FUNCTION "Ventilstatus" : Void
{ S7_Optimized_Access := 'TRUE' }
VERSION : 0.1
   VAR_INPUT 
      SRM_auf : Bool;
      SRM_zu : Bool;
      A_Ventil : Bool;
      Zeit : Time;
   END_VAR

   VAR_OUTPUT 
      "Farbe HMI" : USInt;   // 0: geschlossen (grau) 1: geöffnet (grün) 2: Störung (rot)
      Mld_TO_oeffnen : Bool;
      Mld_TO_schliessen : Bool;
   END_VAR

   VAR_IN_OUT 
      TO_oeffnen {InstructionName := 'TON_TIME'; LibVersion := '1.0'} : TON_TIME;
      TO_schliessen {InstructionName := 'TON_TIME'; LibVersion := '1.0'} : TON_TIME;
      Mld_Sensorfehler : Bool;
   END_VAR

   VAR CONSTANT 
      grau : USInt;
      grün : USInt := 1;
      rot : USInt := 2;
   END_VAR


BEGIN
	// Beide an
	IF #SRM_auf AND #SRM_zu THEN
	    #Mld_Sensorfehler := TRUE;
	ELSIF "DB_ANLAGE".IN.Quitt_Err THEN
	    #Mld_Sensorfehler := FALSE;
	END_IF;
	
	// Zeitüberschreitung öffnen
	#TO_oeffnen(IN := #A_Ventil AND NOT #SRM_auf,
	            PT:= #Zeit,
	            Q=> #Mld_TO_oeffnen);
	
	// Zeitüberschreitung schließen
	#TO_schliessen(IN := NOT #A_Ventil AND NOT #SRM_zu,
	            PT := #Zeit,
	            Q => #Mld_TO_schliessen);
	
	//--> Visu
	IF #Mld_TO_oeffnen OR #Mld_TO_schliessen OR #Mld_Sensorfehler THEN
	    #"Farbe HMI" := #rot;
	ELSIF #A_Ventil THEN
	    #"Farbe HMI" := #grün;
	ELSE
	    #"Farbe HMI" := #grau;
	END_IF;
END_FUNCTION

FUNCTION "Ventilstatus_einfach" : Void
{ S7_Optimized_Access := 'TRUE' }
VERSION : 0.1
   VAR_INPUT 
      A_Ventil : Bool;
   END_VAR

   VAR_OUTPUT 
      "Farbe HMI" : USInt;   // 0: geschlossen (grau) 1: geöffnet (grün) 2: Störung (rot)
   END_VAR

   VAR CONSTANT 
      grau : USInt;
      grün : USInt := 1;
      rot : USInt := 2;
   END_VAR


BEGIN
	//--> Visu
	IF #A_Ventil THEN
	    #"Farbe HMI" := #grün;
	ELSE
	    #"Farbe HMI" := #grau;
	END_IF;
END_FUNCTION

DATA_BLOCK "Deckel_CM01"   // DB1190
// stored: AutoNumber false, InstanceOfName Deckel, InstanceOfType FB
"Deckel"
BEGIN
END_DATA_BLOCK

DATA_BLOCK "Deckel_CM02"   // DB1191
// stored: AutoNumber false, InstanceOfName Deckel, InstanceOfType FB
"Deckel"
BEGIN
END_DATA_BLOCK

DATA_BLOCK "Uhrzeit"   // DB8
// stored: AutoNumber false, InstanceOfName Uhrzeit_WSU, InstanceOfType FB
"Uhrzeit_WSU"
BEGIN
END_DATA_BLOCK

DATA_BLOCK "DI_FU_Fahrt"   // DB181
// stored: AutoNumber false, InstanceOfName FB_FU_OUT_TW, InstanceOfType FB
"FB_FU_OUT_TW"
BEGIN
END_DATA_BLOCK

DATA_BLOCK "DI_FU_Hub_links"   // DB182
// stored: AutoNumber false, InstanceOfName FB_FU_OUT_TW, InstanceOfType FB
"FB_FU_OUT_TW"
BEGIN
END_DATA_BLOCK

DATA_BLOCK "DI_FU_Hub_rechts"   // DB183
// stored: AutoNumber false, InstanceOfName FB_FU_OUT_TW, InstanceOfType FB
"FB_FU_OUT_TW"
BEGIN
END_DATA_BLOCK

DATA_BLOCK "DI_FU_WR02"   // DB184
// stored: AutoNumber false, InstanceOfName FB_FU_OUT_TW, InstanceOfType FB
"FB_FU_OUT_TW"
BEGIN
END_DATA_BLOCK

DATA_BLOCK "DI_FU_WR03"   // DB185
// stored: AutoNumber false, InstanceOfName FB_FU_OUT_TW, InstanceOfType FB
"FB_FU_OUT_TW"
BEGIN
END_DATA_BLOCK

DATA_BLOCK "DI_FW_1"   // DB11
AUTHOR : MS
VERSION : 0.0
// stored: AutoNumber false, InstanceOfName FB_FW_x, InstanceOfType FB
"FB_FW_x"
BEGIN
   Micro.Adr_UP[1] := 16#0066;
   Micro.Adr_UP[2] := 16#006A;
   Micro.Adr_UP[3] := 16#006E;
   Micro.Adr_UP[4] := 16#0077;
   Micro.Adr_UP[5] := 16#007D;
   Micro.Adr_UP[6..13] := 16#0086;
   Micro.Adr_UP[14] := 16#0082;
   Micro.Adr_UP[15] := 16#0084;
   Micro.Liste[0] := 16#02;
   Micro.Liste[1] := 16#14;
   Micro.Liste[2] := 16#05;
   Micro.Liste[3] := 16#00;
   Micro.Liste[4] := 16#03;
   Micro.Liste[5] := 16#14;
   Micro.Liste[6] := 16#05;
   Micro.Liste[7] := 16#00;
   Micro.Liste[8] := 16#01;
   Micro.Liste[9] := 16#15;
   Micro.Liste[10] := 16#04;
   Micro.Liste[11] := 16#0E;
   Micro.Liste[12] := 16#18;
   Micro.Liste[13] := 16#16;
   Micro.Liste[14] := 16#0B;
   Micro.Liste[15] := 16#19;
   Micro.Liste[16] := 16#00;
   Micro.Liste[17] := 16#09;
   Micro.Liste[18] := 16#10;
   Micro.Liste[19] := 16#03;
   Micro.Liste[20] := 16#07;
   Micro.Liste[21] := 16#0C;
   Micro.Liste[22] := 16#00;
   Micro.Liste[23] := 16#14;
   Micro.Liste[24] := 16#09;
   Micro.Liste[25] := 16#11;
   Micro.Liste[26] := 16#12;
   Micro.Liste[27] := 16#00;
   Micro.Liste[28] := 16#0A;
   Micro.Liste[29] := 16#00;
   Micro.Liste[30] := 16#06;
   Micro.Liste[31..79] := 16#00;
END_DATA_BLOCK

DATA_BLOCK "DI_FW_Auftrag_DB"   // DB9
// stored: AutoNumber false, InstanceOfName FB_FW_Auftrag, InstanceOfType FB
"FB_FW_Auftrag"
BEGIN
END_DATA_BLOCK

DATA_BLOCK "DI_FW_HUB_links"   // DB22
AUTHOR : MS
// stored: AutoNumber false, InstanceOfName FB_HUB_FW_li, InstanceOfType FB
"FB_HUB_FW_li"
BEGIN
END_DATA_BLOCK

DATA_BLOCK "DI_FW_HUB_rechts"   // DB23
AUTHOR : MS
// stored: AutoNumber false, InstanceOfName FB_HUB_FW_re, InstanceOfType FB
"FB_HUB_FW_re"
BEGIN
END_DATA_BLOCK

DATA_BLOCK "DI_FW_MANAGER"   // DB10
AUTHOR : MS
// stored: AutoNumber false, InstanceOfName FB_FW_MANAGER, InstanceOfType FB
"FB_FW_MANAGER"
BEGIN
   Kettenpos[1..4] := 16#00;
   FW_DAT[1..20].WT_NR_LANG := 0;
   FW_DAT[1].IST_POS := 16#02;
   FW_DAT[2].IST_POS := 16#0B;
   FW_DAT[3].IST_POS := 16#2C;
   FW_DAT[4].IST_POS := 16#4A;
   FW_DAT[5].IST_POS := 16#02;
   FW_DAT[6].IST_POS := 16#2F;
   FW_DAT[7..20].IST_POS := 16#00;
   FW_DAT[1..20].ZIEL_POS := 16#00;
   FW_DAT[1..20].Fahrt_Vor := FALSE;
   FW_DAT[1..20].Fahrt_Rck := FALSE;
   FW_DAT[1..20].Heben := FALSE;
   FW_DAT[1..20].Senken := FALSE;
   FW_DAT[1..6].Bereit := TRUE;
   FW_DAT[7..20].Bereit := FALSE;
   FW_DAT[1..20].Fehler := FALSE;
   FW_DAT[1..20].Dummy := FALSE;
   FW_DAT[1..20].res := FALSE;
   FW_DAT[1..20].Tipp := FALSE;
   FW_DAT[1..6].Hand := TRUE;
   FW_DAT[7..20].Hand := FALSE;
   FW_DAT[1..20].Auto_Stop := FALSE;
   FW_DAT[1..20].Auto := FALSE;
   FW_DAT[1..20].Halt := FALSE;
   FW_DAT[1..6].K_Auto := TRUE;
   FW_DAT[7..20].K_Auto := FALSE;
   FW_DAT[1..4].Kette_wait_Start := TRUE;
   FW_DAT[5..20].Kette_wait_Start := FALSE;
   FW_DAT[1..4].Kette_wait_Ende := TRUE;
   FW_DAT[5..20].Kette_wait_Ende := FALSE;
   FW_DAT[1..4].Unten := TRUE;
   FW_DAT[5..20].Unten := FALSE;
   FW_DAT[1..20].Z_Sensor := FALSE;
   FW_DAT[1..20].Oben := FALSE;
   FW_DAT[1..6].mittig := TRUE;
   FW_DAT[7..20].mittig := FALSE;
   FW_DAT[1..20].HWmittig := FALSE;
   FW_DAT[1..20].res_7 := FALSE;
   FW_DAT[1..20].res_8 := FALSE;
   FW_DAT[1..20].res_9 := FALSE;
   FW_DAT[1..20].WT_DB_Nr := 16#00;
   FW_DAT[1].IstInc := 1998;
   FW_DAT[2].IstInc := 10998;
   FW_DAT[3].IstInc := 43999;
   FW_DAT[4].IstInc := 49759;
   FW_DAT[5..20].IstInc := 0;
   FW_DAT[1..20].Stangen_Nr := 16#00;
   FW_DAT[1..20].WT_Typ := 16#00;
   FW_DAT[1..20].priorisirt := FALSE;
   FW_DAT[1..20].in_Anlage := FALSE;
   FW_DAT[1..20].in_Entmetall := FALSE;
   FW_DAT[1..20].aus_Anlage := FALSE;
   FW_DAT[1..20].aus_Entmetall := FALSE;
   FW_DAT[1..20].Speicherprog := FALSE;
   FW_DAT[1..20].Trommel := FALSE;
   FW_DAT[1..20].Leer_WT := FALSE;
   FW_DAT[1..20].BefX := 16#00;
END_DATA_BLOCK

DATA_BLOCK "DI_FW_POS_1"   // DB21
// stored: AutoNumber false, InstanceOfName FB_POS_FW_INC, InstanceOfType FB
"FB_POS_FW_INC"
BEGIN
END_DATA_BLOCK

DATA_BLOCK "DI_QF_WR02_03"   // DB31
// stored: AutoNumber false, InstanceOfName FB_QF, InstanceOfType FB
"FB_QF"
BEGIN
END_DATA_BLOCK

DATA_BLOCK "Tor"   // DB1092
// stored: AutoNumber false, InstanceOfName RT, InstanceOfType FB
"RT"
BEGIN
END_DATA_BLOCK

DATA_BLOCK "TCON_DI"   // DB365
// stored: AutoNumber false, InstanceOfName TCON, OfSystemLibElement TCON, OfSystemLibVersion 4.0
"TCON"
   // VAR_INPUT
   //    REQ : Bool := TRUE;
   //    ID : CONN_OUC := 16#0002;
   // END_VAR
   // VAR_OUTPUT
   //    DONE : Bool := TRUE;
   //    BUSY : Bool := FALSE;
   //    ERROR : Bool := FALSE;
   //    STATUS : Word := 16#0000;
   // END_VAR
   // VAR_IN_OUT
   //    CONNECT : Variant;
   // END_VAR
BEGIN
END_DATA_BLOCK

DATA_BLOCK "TDISCON_DI"   // DB368
// stored: AutoNumber false, InstanceOfName T_DISCON, OfSystemLibElement TDISCON, OfSystemLibVersion 2.1
"T_DISCON"
   // VAR_INPUT
   //    REQ : Bool := FALSE;
   //    ID : CONN_OUC := 16#0000;
   // END_VAR
   // VAR_OUTPUT
   //    DONE : Bool := FALSE;
   //    BUSY : Bool := FALSE;
   //    ERROR : Bool := FALSE;
   //    STATUS : Word := 16#7000;
   // END_VAR
BEGIN
END_DATA_BLOCK

DATA_BLOCK "TRCV_DI"   // DB367
// stored: AutoNumber false, InstanceOfName TRCV, OfSystemLibElement TRCV, OfSystemLibVersion 4.0
"TRCV"
   // VAR_INPUT
   //    EN_R : Bool := TRUE;
   //    ID : CONN_OUC := 16#0002;
   //    LEN : UDInt := 30;
   //    ADHOC : Bool := FALSE;
   // END_VAR
   // VAR_OUTPUT
   //    NDR : Bool := TRUE;
   //    BUSY : Bool := FALSE;
   //    ERROR : Bool := FALSE;
   //    STATUS : Word := 16#0000;
   //    RCVD_LEN : UDInt := 30;
   // END_VAR
   // VAR_IN_OUT
   //    DATA : Variant;
   //    ADDR : Variant;
   // END_VAR
BEGIN
END_DATA_BLOCK

DATA_BLOCK "TSEND_DI"   // DB366
// stored: AutoNumber false, InstanceOfName TSEND, OfSystemLibElement TSEND, OfSystemLibVersion 4.0
"TSEND"
   // VAR_INPUT
   //    REQ : Bool := TRUE;
   //    ID : CONN_OUC := 16#0002;
   //    LEN : UDInt := 30;
   // END_VAR
   // VAR_OUTPUT
   //    DONE : Bool := TRUE;
   //    BUSY : Bool := FALSE;
   //    ERROR : Bool := FALSE;
   //    STATUS : Word := 16#0000;
   // END_VAR
   // VAR_IN_OUT
   //    DATA : Variant;
   //    ADDR : Variant;
   // END_VAR
BEGIN
END_DATA_BLOCK

DATA_BLOCK "FP_CM01.GP01"   // DB1001
// stored: AutoNumber false, InstanceOfName FP_Saeure.GP0x, InstanceOfType FB
"FP_Saeure.GP0x"
BEGIN
END_DATA_BLOCK

DATA_BLOCK "FP_CM02.GP04"   // DB1004
// stored: AutoNumber false, InstanceOfName FP_Saeure.GP0x, InstanceOfType FB
"FP_Saeure.GP0x"
BEGIN
END_DATA_BLOCK

DATA_BLOCK "Pu_CL01.GP08"   // DB1008
// stored: AutoNumber false, InstanceOfName Pu_Entl.GP0x, InstanceOfType FB
"Pu_Entl.GP0x"
BEGIN
END_DATA_BLOCK

DATA_BLOCK "Pu_CL02.GP09"   // DB1009
// stored: AutoNumber false, InstanceOfName Pu_Entl.GP0x, InstanceOfType FB
"Pu_Entl.GP0x"
BEGIN
END_DATA_BLOCK

DATA_BLOCK "Pu_CM05.GP11_DB"   // DB1011
// stored: AutoNumber false, InstanceOfName Pu_CM05.GP11, InstanceOfType FB
"Pu_CM05.GP11"
BEGIN
END_DATA_BLOCK

DATA_BLOCK "Pu_GP01.GP12"   // DB1012
// stored: AutoNumber false, InstanceOfName Pu_Entl.GP0x, InstanceOfType FB
"Pu_Entl.GP0x"
BEGIN
END_DATA_BLOCK

DATA_BLOCK "Pu_GP01.GP13"   // DB1013
// stored: AutoNumber false, InstanceOfName Pu_Versorgung.GP0x, InstanceOfType FB
"Pu_Versorgung.GP0x"
BEGIN
END_DATA_BLOCK

DATA_BLOCK "Pu_GP02.GP07"   // DB1007
// stored: AutoNumber false, InstanceOfName Pu_Entl.GP0x, InstanceOfType FB
"Pu_Entl.GP0x"
BEGIN
END_DATA_BLOCK

DATA_BLOCK "Pu_GP02.GP10"   // DB1010
// stored: AutoNumber false, InstanceOfName Pu_Versorgung.GP0x, InstanceOfType FB
"Pu_Versorgung.GP0x"
BEGIN
END_DATA_BLOCK

DATA_BLOCK "UP_CM01.GP02"   // DB1002
// stored: AutoNumber false, InstanceOfName UP_Saeure.GP0x, InstanceOfType FB
"UP_Saeure.GP0x"
BEGIN
END_DATA_BLOCK

DATA_BLOCK "UP_CM02.GP05"   // DB1005
// stored: AutoNumber false, InstanceOfName UP_Saeure.GP0x, InstanceOfType FB
"UP_Saeure.GP0x"
BEGIN
END_DATA_BLOCK

DATA_BLOCK "UP_CM03.GP03"   // DB1003
// stored: AutoNumber false, InstanceOfName UP_Spuele.GP0x, InstanceOfType FB
"UP_Spuele.GP0x"
BEGIN
END_DATA_BLOCK

DATA_BLOCK "UP_CM04.GP06"   // DB1006
// stored: AutoNumber false, InstanceOfName UP_Spuele.GP0x, InstanceOfType FB
"UP_Spuele.GP0x"
BEGIN
END_DATA_BLOCK

DATA_BLOCK "Ventil_Stati_DB"   // DB1095
// stored: AutoNumber false, InstanceOfName Ventil_Stati, InstanceOfType FB
"Ventil_Stati"
BEGIN
END_DATA_BLOCK
